FUNCTION_BLOCK ExtractiveOutletHandler
VAR_INPUT
	stop : BOOL;
	extractiveControlValveCommands : ST_ExtractiveControlValveCommands;
	extractiveControlValveParameters : ST_ExtractiveControlValveParameters;
	extractiveOutOnOffValveCommand : BOOL;
	autoExtractionControlValveValue : DINT;
	autoExtractionStarted : BOOL;
END_VAR
VAR_OUTPUT
	extractiveOnOffValveValues : ST_ExtractiveOnOffValveValues;
	controlValveOpeningPercentage : DINT;
	calibrateDone : BOOL;
	openOnOffValve : BOOL;
	closeExtractiveOutletValve : BOOL;
	openExtractiveOutletValve : BOOL;
END_VAR
VAR
	pressureReference : INT;
	ExtractiveOutletControl : FB_ExtractiveOutletControl;
END_VAR


extractiveControlValveCommands.stopCalibration := stop;

IF autoExtractionStarted THEN
	extractiveControlValveCommands.openPercentage := autoExtractionControlValveValue;
END_IF

ExtractiveOutletControl(
					onOffValveCommand := extractiveOutOnOffValveCommand,
					controlValveCommands := extractiveControlValveCommands,
					controlValveParameters := extractiveControlValveParameters,
					onOffValveOpen => ,
					onOffValveButtonCommand => openOnOffValve,//GVL_IO.extractiveOutletOnOffValve,
					controlValveClose => closeExtractiveOutletValve,
					controlValveOpen => openExtractiveOutletValve,
					controlValveCurrentOpenPercentage => controlValveOpeningPercentage,
					calibrateDone => calibrateDone);
					
extractiveOnOffValveValues.open := ExtractiveOutletControl.onOffValveOpen;

END_FUNCTION_BLOCK

(* stored: Version 1.1.0.1, ProductVersion 3.1.4024.9
   POU ExtractiveOutletHandler: Id {cb9f01f2-17f8-480e-83e5-bbdc38e2f096}, SpecialFunc None *)
